// Mitsubishi GX Works2 project: stepper   PLC: FX1S

PROGRAM MAIN
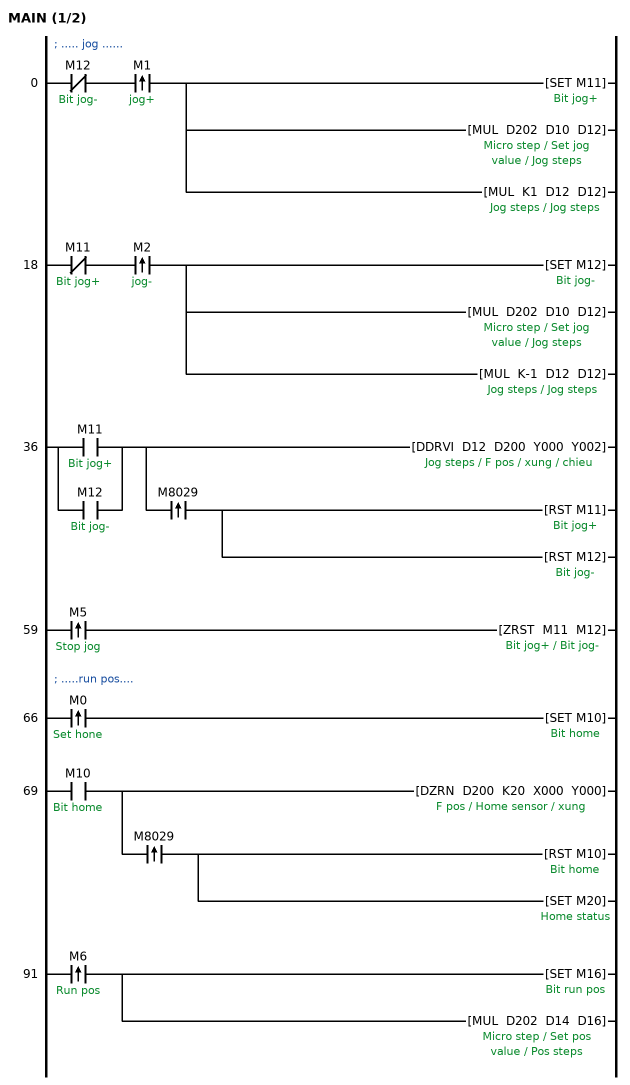
; ..... jog ......
0     LDI     M12  ; Bit jog-
      ANDP    M1  ; jog+
      SET     M11  ; Bit jog+
      MUL     D202 D10 D12  ; Micro step / Set jog value / Jog steps
      MUL     K1 D12 D12
18    LDI     M11  ; Bit jog+
      ANDP    M2  ; jog-
      SET     M12  ; Bit jog-
      MUL     D202 D10 D12
      MUL     K-1 D12 D12
36    LD      M11  ; Bit jog+
      OR      M12  ; Bit jog-
      DDRVI   D12 D200 Y000 Y002  ; F pos / xung / chieu
      ANDP    M8029
      RST     M11  ; Bit jog+
      RST     M12  ; Bit jog-
59    LDP     M5  ; Stop jog
      ZRST    M11 M12
; .....run pos....
66    LDP     M0  ; Set hone
      SET     M10  ; Bit home
69    LD      M10  ; Bit home
      DZRN    D200 K20 X000 Y000  ; Home sensor
      ANDP    M8029
      RST     M10  ; Bit home
      SET     M20  ; Home status
; 
91    LDP     M6  ; Run pos
      SET     M16  ; Bit run pos
      MUL     D202 D14 D16  ; Set pos value / Pos steps
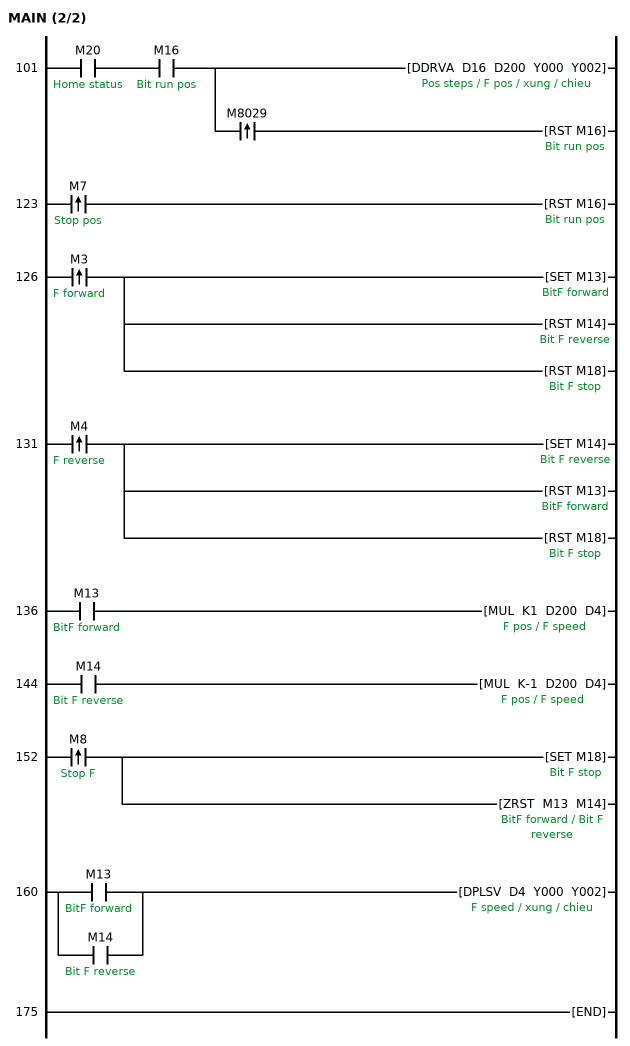
101   LD      M20  ; Home status
      AND     M16  ; Bit run pos
      DDRVA   D16 D200 Y000 Y002
      ANDP    M8029
      RST     M16  ; Bit run pos
123   LDP     M7  ; Stop pos
      RST     M16  ; Bit run pos
126   LDP     M3  ; F forward
      SET     M13  ; BitF forward
      RST     M14  ; Bit F reverse
      RST     M18  ; Bit F stop
131   LDP     M4  ; F reverse
      SET     M14  ; Bit F reverse
      RST     M13  ; BitF forward
      RST     M18  ; Bit F stop
136   LD      M13  ; BitF forward
      MUL     K1 D200 D4  ; F speed
144   LD      M14  ; Bit F reverse
      MUL     K-1 D200 D4
152   LDP     M8  ; Stop F
      SET     M18  ; Bit F stop
      ZRST    M13 M14
160   LD      M13  ; BitF forward
      OR      M14  ; Bit F reverse
      DPLSV   D4 Y000 Y002
175   END
END_PROGRAM

// device comments not shown above
Y003  ; enable
M17  ; Bit stop pos
